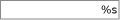
VISUALIZATION visUINT_QUERRY  // 120x20
VAR_INPUT
    visfbUINTIn :   ITF_UINT;	
END_VAR
VAR_INPUT 
    stPhysikalischeEinheit  : STRING[5];
END_VAR
    Frame (0,0 120x20), invisible if: NOT __QUERYINTERFACE(visfbUINTIn,visfbUINTIn)
        shows visUINT_ITF(visfbUINT := visfbUINTIn, stPhysikalischeEinheit := stPhysikalischeEinheit)
END_VISUALIZATION

// 40 Visualizations/32 Bit/DWORD/visDWORD_ITF
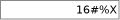
VISUALIZATION visDWORD_ITF  // 120x20
VAR_INPUT
    visfbDWORD   :   ITF_DWORD;	
END_VAR
    Textfield (0,0 120x20), "16#%X", text variable: visfbDWORD.proValue
        OnMouseClick: write the text variable via InputWithLimits, min visfbDWORD.proMin, max visfbDWORD.proMax
END_VISUALIZATION

// 40 Visualizations/8 Bit/BYTE/visBYTE_QUERRY
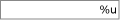
VISUALIZATION visBYTE_QUERRY  // 120x20
VAR_INPUT
    visfbBYTEIn :   ITF_BYTE;	
END_VAR
    Frame (0,0 120x20), invisible if: NOT __QUERYINTERFACE(visfbBYTEIn,visfbBYTEIn)
        shows visBYTE_ITF(visfbBYTE := visfbBYTEIn)
END_VISUALIZATION

// 40 Visualizations/32 Bit/UDINT/visUDINT_ITF
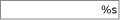
VISUALIZATION visUDINT_ITF  // 120x20
VAR_INPUT
    visfbUDINT   :   ITF_UDINT;	
END_VAR
VAR_INPUT 
    stPhysikalischeEinheit  : STRING[5];
END_VAR
    Textfield (0,0 120x20), "%s", text variable: CONCAT(TO_STRING(visfbUDINT.proValue),stPhysikalischeEinheit)
        OnMouseClick: write visfbUDINT.proValue via InputWithLimits, min visfbUDINT.proMin, max visfbUDINT.proMax
END_VISUALIZATION

// 40 Visualizations/16 Bit/WORD/WORD HEX/visWORD_ITF_HEX
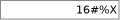
VISUALIZATION visWORD_ITF_HEX  // 120x20
VAR_INPUT
    visfbWORD   :   ITF_WORD;	
END_VAR
    Textfield (0,0 120x20), "16#%X", text variable: visfbWORD.proValue
        OnMouseClick: write the text variable via InputWithLimits, min visfbWORD.proMin, max visfbWORD.proMax
END_VISUALIZATION

// 40 Visualizations/8 Bit/SINT/visSINT
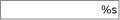
VISUALIZATION visSINT  // 120x20
VAR_INPUT
    visfbSINTIn :   ITF_DATATYPE;	
END_VAR
VAR
    visfbSINT   :   ITF_SINT;	
END_VAR
VAR_INPUT 
    stPhysikalischeEinheit  : STRING[5];
END_VAR
    Frame (0,0 120x20), invisible if: NOT __QUERYINTERFACE(visfbSINTIn,visfbSINT)
        shows visSINT_QUERRY(visfbSINTIn := visfbSINT, stPhysikalischeEinheit := stPhysikalischeEinheit)
END_VISUALIZATION

// 40 Visualizations/Show Data/visSHOWDATA_ITF
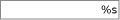
VISUALIZATION visSHOWDATA_ITF  // 120x20
VAR_INPUT
    visfbDATATYPEIn     :   ITF_DATATYPE;	
END_VAR
VAR_INPUT 
    stPhysikalischeEinheit  : STRING[5];
END_VAR
    Textfield (0,0 120x20), "%s", text variable: CONCAT(visfbDATATYPEIn.proShowValue,CONCAT(' ',stPhysikalischeEinheit))
END_VISUALIZATION

// 40 Visualizations/8 Bit/USINT/visUSINT
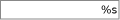
VISUALIZATION visUSINT  // 120x20
VAR_INPUT
    visfbUSINTIn :   ITF_DATATYPE;	
END_VAR
VAR
    visfbUSINT   :   ITF_USINT;	
END_VAR
VAR_INPUT 
    stPhysikalischeEinheit  : STRING[5];
END_VAR
    Frame (0,0 120x20), invisible if: NOT __QUERYINTERFACE(visfbUSINTIn,visfbUSINT)
        shows visUSINT_QUERRY(visfbUSINTIn := visfbUSINT, stPhysikalischeEinheit := stPhysikalischeEinheit)
END_VISUALIZATION

// 40 Visualizations/32 Bit/REAL/visREAL_ITF
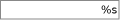
VISUALIZATION visREAL_ITF  // 120x20
VAR_INPUT    
    visfbREAL   :   ITF_REAL;	
END_VAR
VAR_INPUT 
    stPhysikalischeEinheit  : STRING[5];
END_VAR
    Textfield (0,0 120x20), "%s", text variable: CONCAT(fcRealToString(visfbREAL.proValue,2),stPhysikalischeEinheit)
        OnMouseClick: write visfbREAL.proValue via InputWithLimits, min visfbREAL.proMin, max visfbREAL.proMax
END_VISUALIZATION

// 40 Visualizations/64 Bit/LTIME/visLTIME_QUERRY
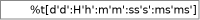
VISUALIZATION visLTIME_QUERRY  // 200x20
VAR_INPUT
    visfbLTIMEIn :   ITF_LTIME;	
END_VAR
    Frame (0,0 200x20), invisible if: NOT __QUERYINTERFACE(visfbLTIMEIn,visfbLTIMEIn)
        shows visLTIME_ITF(visfbLTIME := visfbLTIMEIn)
END_VISUALIZATION

// 40 Visualizations/32 Bit/DWORD/visDWORD
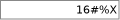
VISUALIZATION visDWORD  // 120x20
VAR_INPUT
    visfbDWORDIn :   ITF_DATATYPE;	
END_VAR
VAR
    visfbDWORD   :   ITF_DWORD;	
END_VAR
    Frame (0,0 120x20), invisible if: NOT __QUERYINTERFACE(visfbDWORDIn,visfbDWORD)
        shows visDWORD_QUERRY(visfbDWORDIn := visfbDWORD)
END_VISUALIZATION

// 40 Visualizations/ENUMERATION/8 Bit/visENUMERATION_BYTE
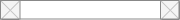
VISUALIZATION visENUMERATION_BYTE  // 180x20
VAR_INPUT
    visfbBYTE   :   ITF_BYTE;		
END_VAR
    Image (160,0 20x20), image: CtaVisSymbols.ImagePool.arrow-right_square
        OnMouseClick: execute {
            IF visfbBYTE.proValue < visfbBYTE.proMax THEN
                visfbBYTE.proValue := visfbBYTE.proValue + 1;
            ELSIF visfbBYTE.proValue = visfbBYTE.proMax THEN
                visfbBYTE.proValue := visfbBYTE.proMin;
            END_IF;
        }
    Image (0,0 20x20), image: CtaVisSymbols.ImagePool.arrow-left_square
        OnMouseClick: execute {
            IF visfbBYTE.proValue > visfbBYTE.proMin THEN
                visfbBYTE.proValue := visfbBYTE.proValue - 1;
            ELSIF visfbBYTE.proValue = visfbBYTE.proMin THEN
                visfbBYTE.proValue := visfbBYTE.proMax;
            END_IF;
        }
END_VISUALIZATION

// 40 Visualizations/ENUMERATION/8 Bit/visENUMERATION_BYTE_QUERR
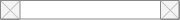
VISUALIZATION visENUMERATION_BYTE_QUERR  // 180x20
VAR_INPUT
    visfbBYTE   :   ITF_BYTE;	
END_VAR
    Frame (0,0 180x20), invisible if: NOT __QUERYINTERFACE(visfbBYTE,visfbBYTE)
        shows visENUMERATION_BYTE(visfbBYTE := visfbBYTE)
END_VISUALIZATION
